// TwinCAT 3 PLC project FMS_201_Estructurado
// ProgramVersion: 3.1.4024.0
// libraries:
//   Tc2_Standard, * (Beckhoff Automation GmbH)
//   Tc2_System, * (Beckhoff Automation GmbH)
//   Tc3_Module, * (Beckhoff Automation GmbH)
// project tree:
//   / PlcTask.TcTTO (not stored)
//   POUs/Estación/ FB_Coordinador_SFC.TcPOU (not stored), FB_Estacion_SFC.TcPOU (not stored)
//   POUs/ MAIN.TcPOU
//   POUs/Tareas/ FB_2_AlimentarBase_SFC.TcPOU, FB_1_CargarBase_SFC.TcPOU (not stored), FB_4_InsertarBasePale_SFCC.TcPOU, FB_5_TransferirBase_SFC.TcPOU, FB_3_VerificarPale_SFC.TcPOU
// (motion and I/O tree: see PLC project fms_201_manual)
// real-time tasks:
//   TASK PlcTask: cycle T#10ms, priority 20, ADS port 350
//   TASK PlcTask1: cycle T#10ms, priority 21, ADS port 351
//   TASK PlcTask2: cycle T#10ms, priority 22, ADS port 352
//   TASK PlcTask3: cycle T#10ms, priority 23, ADS port 353
//   TASK PlcTask4: cycle T#10ms, priority 24, ADS port 354
//   TASK PlcTask5: cycle T#10ms, priority 25, ADS port 355
//   TASK PlcTask6: cycle T#10ms, priority 26, ADS port 356
// variable links:

// ---- POUs/MAIN.TcPOU
PROGRAM MAIN
VAR
END_VAR

END_PROGRAM

// ---- POUs/Tareas/FB_2_AlimentarBase_SFC.TcPOU
FUNCTION_BLOCK FB_2_AlimentarBase_SFC
VAR_INPUT
	
	//  SFC-Flags
	SFCPause: BOOL;
	SFCReset: BOOL;

	// Indicadores de sincronización
	Ack: BOOL := TRUE;
	Execute: BOOL;
	
	// Entradas
	AlimentadorDetras: BOOL;
	AlimentadorDelante: BOOL;
	PresenciaBaseAlimentador: BOOL;
	PulsadorMarcha: BOOL;
	
END_VAR
VAR_OUTPUT
	
	// Indicadores de sincronización
	Ready: BOOL;	
	Done: BOOL;
	
	// Salidas
	AlimentadorAdelante: BOOL;
	LamparaFaltaMaterial: BOOL;
	
END_VAR
VAR
END_VAR

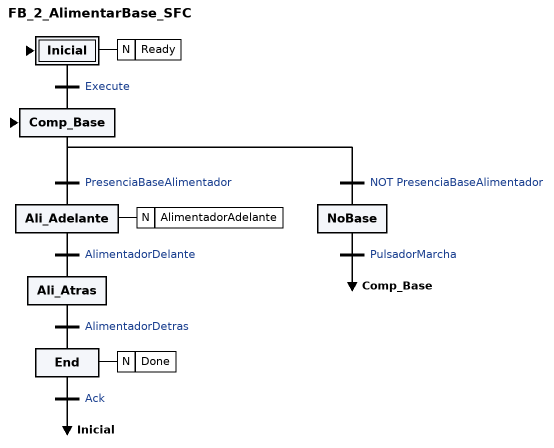
INITIAL_STEP Inicial:
    Ready(N);
END_STEP
TRANSITION FROM Inicial TO Comp_Base
    := Execute;
END_TRANSITION
STEP Comp_Base:
END_STEP
TRANSITION FROM Comp_Base TO Ali_Adelante
    := PresenciaBaseAlimentador;
END_TRANSITION
TRANSITION FROM Comp_Base TO NoBase
    := NOT PresenciaBaseAlimentador;
END_TRANSITION
STEP NoBase:
END_STEP
TRANSITION FROM NoBase TO Comp_Base
    := PulsadorMarcha;
END_TRANSITION
STEP Ali_Adelante:
    AlimentadorAdelante(N);
END_STEP
TRANSITION FROM Ali_Adelante TO Ali_Atras
    := AlimentadorDelante;
END_TRANSITION
STEP Ali_Atras:
END_STEP
TRANSITION FROM Ali_Atras TO End
    := AlimentadorDetras;
END_TRANSITION
STEP End:
    Done(N);
END_STEP
TRANSITION FROM End TO Inicial
    := Ack;
END_TRANSITION

END_FUNCTION_BLOCK

// ---- POUs/Tareas/FB_4_InsertarBasePale_SFCC.TcPOU
FUNCTION_BLOCK FB_4_InsertarBasePale_SFCC
VAR_INPUT

	//  SFC-Flags
	SFCPause: BOOL;
	SFCReset: BOOL;

	// Indicadores de sincronización
	Ack: BOOL := TRUE;
	Execute: BOOL;
	
	// Entradas
	VerticalArriba: BOOL;
	VerticalAbajo: BOOL;
	VacioDescargador: BOOL;	
	DescargadorDetras: BOOL;
	DescargadorDelante: BOOL;
	
END_VAR
VAR_OUTPUT
	
// Indicadores de sincronización
	Ready: BOOL;	
	Done: BOOL;
	
	// Salidas
	DescargadorAtras: BOOL;
	DescargadorAdelante: BOOL;
	DescargadorBaja : BOOL;
	EyectorSucciona : BOOL;
	
END_VAR
VAR
END_VAR

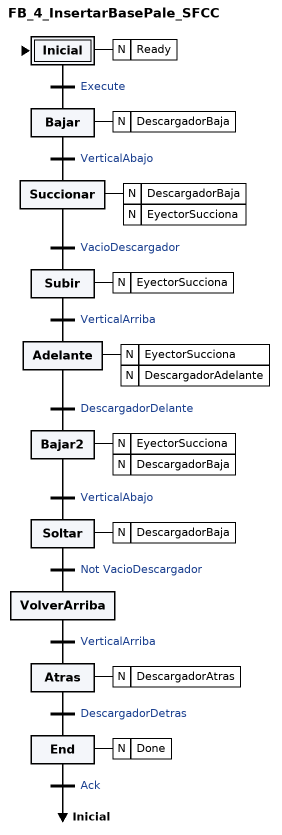
INITIAL_STEP Inicial:
    Ready(N);
END_STEP
TRANSITION FROM Inicial TO Bajar
    := Execute;
END_TRANSITION
STEP Bajar:
    DescargadorBaja(N);
END_STEP
TRANSITION FROM Bajar TO Succionar
    := VerticalAbajo;
END_TRANSITION
STEP Succionar:
    DescargadorBaja(N);
    EyectorSucciona(N);
END_STEP
TRANSITION FROM Succionar TO Subir
    := VacioDescargador;
END_TRANSITION
STEP Subir:
    EyectorSucciona(N);
END_STEP
TRANSITION FROM Subir TO Adelante
    := VerticalArriba;
END_TRANSITION
STEP Adelante:
    EyectorSucciona(N);
    DescargadorAdelante(N);
END_STEP
TRANSITION FROM Adelante TO Bajar2
    := DescargadorDelante;
END_TRANSITION
STEP Bajar2:
    EyectorSucciona(N);
    DescargadorBaja(N);
END_STEP
TRANSITION FROM Bajar2 TO Soltar
    := VerticalAbajo;
END_TRANSITION
STEP Soltar:
    DescargadorBaja(N);
END_STEP
TRANSITION FROM Soltar TO VolverArriba
    := Not VacioDescargador;
END_TRANSITION
STEP VolverArriba:
END_STEP
TRANSITION FROM VolverArriba TO Atras
    := VerticalArriba;
END_TRANSITION
STEP Atras:
    DescargadorAtras(N);
END_STEP
TRANSITION FROM Atras TO End
    := DescargadorDetras;
END_TRANSITION
STEP End:
    Done(N);
END_STEP
TRANSITION FROM End TO Inicial
    := Ack;
END_TRANSITION

END_FUNCTION_BLOCK

// ---- POUs/Tareas/FB_5_TransferirBase_SFC.TcPOU
FUNCTION_BLOCK FB_5_TransferirBase_SFC
VAR_INPUT
	
	//  SFC-Flags
	SFCPause: BOOL;
	SFCReset: BOOL;

	// Indicadores de sincronización
	Ack: BOOL := TRUE;
	Execute: BOOL;
	
	// Entradas
	PalePresencia: BOOL;
	TpoCintaFuera: TIME;
	TpoRetenedorBaja: TIME;
	
END_VAR
VAR_OUTPUT
	
	// Indicadores de sincronización
	Ready: BOOL;	
	Done: BOOL;
	
	// Salidas
	CintaMotorActiva: BOOL;
	CintaRetenedorBaja: BOOL;
	CintaSeparadorSube: BOOL;
	
END_VAR
VAR
END_VAR

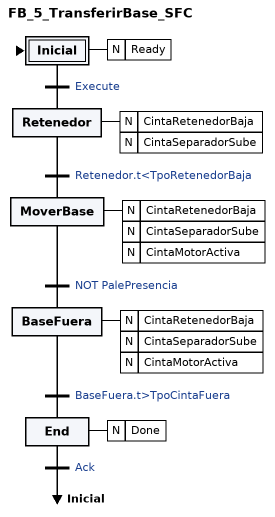
INITIAL_STEP Inicial:
    Ready(N);
END_STEP
TRANSITION FROM Inicial TO Retenedor
    := Execute;
END_TRANSITION
STEP Retenedor:
    CintaRetenedorBaja(N);
    CintaSeparadorSube(N);
END_STEP
TRANSITION FROM Retenedor TO MoverBase
    := Retenedor.t<TpoRetenedorBaja;
END_TRANSITION
STEP MoverBase:
    CintaRetenedorBaja(N);
    CintaSeparadorSube(N);
    CintaMotorActiva(N);
END_STEP
TRANSITION FROM MoverBase TO BaseFuera
    := NOT PalePresencia;
END_TRANSITION
STEP BaseFuera:
    CintaRetenedorBaja(N);
    CintaSeparadorSube(N);
    CintaMotorActiva(N);
END_STEP
TRANSITION FROM BaseFuera TO End
    := BaseFuera.t>TpoCintaFuera;
END_TRANSITION
STEP End:
    Done(N);
END_STEP
TRANSITION FROM End TO Inicial
    := Ack;
END_TRANSITION

END_FUNCTION_BLOCK

// ---- POUs/Tareas/FB_3_VerificarPale_SFC.TcPOU
FUNCTION_BLOCK FB_3_VerificarPale_SFC
VAR_INPUT
	
	//  SFC-Flags
	SFCPause: BOOL;
	SFCReset: BOOL;

	// Indicadores de sincronización
	Ack: BOOL := TRUE;
	Execute: BOOL;
	
	// Entradas
	VerificadorAbajo: BOOL;
	VerificadorArriba: BOOL;
	DesplazadorDetras: BOOL;
	TpoVerificador: TIME;
	TpoDesplazador: TIME;
	TpoRechazador: TIME;
	
END_VAR
VAR_OUTPUT
	
	// Indicadores de sincronización
	Ready: BOOL;	
	Done: BOOL;
	DoneIncorrecto: BOOL;
	// Salidas
	VerificadorBaja: BOOL;
	DesplazadorAdelante: BOOL;
	RechazadorAdelante: BOOL;
	
END_VAR

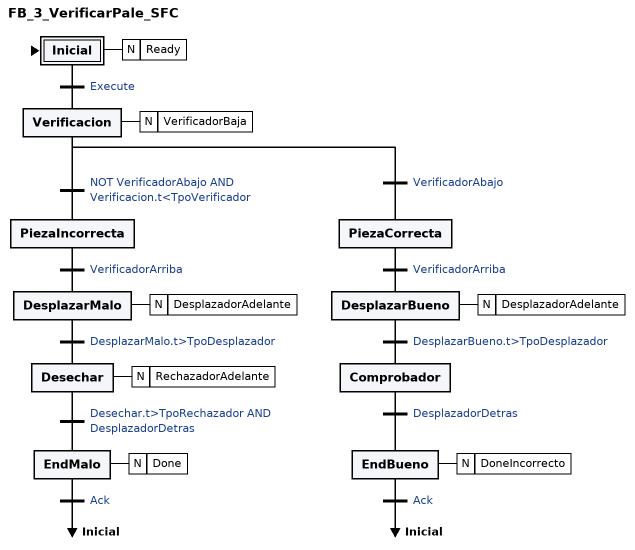
INITIAL_STEP Inicial:
    Ready(N);
END_STEP
TRANSITION FROM Inicial TO Verificacion
    := Execute;
END_TRANSITION
STEP Verificacion:
    VerificadorBaja(N);
END_STEP
TRANSITION FROM Verificacion TO PiezaIncorrecta
    := NOT VerificadorAbajo AND Verificacion.t<TpoVerificador;
END_TRANSITION
STEP PiezaIncorrecta:
END_STEP
TRANSITION FROM PiezaIncorrecta TO DesplazarMalo
    := VerificadorArriba;
END_TRANSITION
STEP DesplazarMalo:
    DesplazadorAdelante(N);
END_STEP
TRANSITION FROM DesplazarMalo TO Desechar
    := DesplazarMalo.t>TpoDesplazador;
END_TRANSITION
STEP Desechar:
    RechazadorAdelante(N);
END_STEP
TRANSITION FROM Desechar TO EndMalo
    := Desechar.t>TpoRechazador AND DesplazadorDetras;
END_TRANSITION
STEP EndMalo:
    Done(N);
END_STEP
TRANSITION FROM EndMalo TO Inicial
    := Ack;
END_TRANSITION
TRANSITION FROM Verificacion TO PiezaCorrecta
    := VerificadorAbajo;
END_TRANSITION
STEP PiezaCorrecta:
END_STEP
TRANSITION FROM PiezaCorrecta TO DesplazarBueno
    := VerificadorArriba;
END_TRANSITION
STEP DesplazarBueno:
    DesplazadorAdelante(N);
END_STEP
TRANSITION FROM DesplazarBueno TO Comprobador
    := DesplazarBueno.t>TpoDesplazador;
END_TRANSITION
STEP Comprobador:
END_STEP
TRANSITION FROM Comprobador TO EndBueno
    := DesplazadorDetras;
END_TRANSITION
STEP EndBueno:
    DoneIncorrecto(N);
END_STEP
TRANSITION FROM EndBueno TO Inicial
    := Ack;
END_TRANSITION

END_FUNCTION_BLOCK
